(* LS Electric XG5000 project: InchingWalkThroughEX *)
(* PLC LSPLC *)
(* module base 0 slot 0: Input/Output Module:XEM-DN/DP32HP (DC 24V Input, Transistor Output, 32 Contacts) *)
(* module base 0 slot 1: Internal Positioning:XBF-PO06E (Open Collector Type, 6 Axis) *)

(* Comments on direct variables
%IX0.0.4	Jog FWD Ax1
%IX0.0.5	Jog REV Ax1
*)

PROGRAM Jog (* task: Scan Program *)
VAR
    Axis1_Inch_FWD : APM_INC;
    Axis1_Inch_FWD1 : XPM_INC;
    Axis1_Inch_REV : XPM_INC;
    Axis1_Jog_FWD : XPM_JOG;
    Axis1_Jog_REV : XPM_JOG;
    AXIS1_RST : XPM_RST;
    Axis1_RTP : XPM_RTP;
    Axis1_STP : XPM_STP;
END_VAR

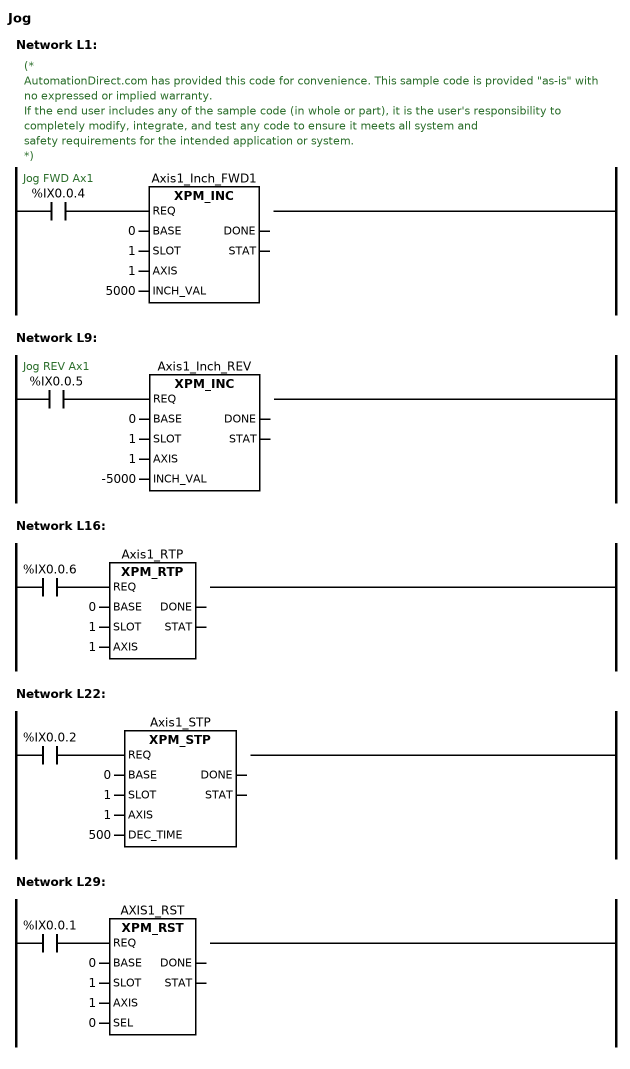
(* ( * / AutomationDirect.com has provided this code for convenience. This sample code is provided "as-is" with no expressed or implied warranty. / If the end user includes any of the sample code (in whole or part), it is the user's responsibility to completely modify, integrate, and test any code to ensure it meets all system and / safety requirements for the intended application or system. / * ) *)
(* Rung L1 *)
Axis1_Inch_FWD1(REQ := %IX0.0.4, BASE := 0, SLOT := 1, AXIS := 1, INCH_VAL := 5000);
(* Rung L9 *)
Axis1_Inch_REV(REQ := %IX0.0.5, BASE := 0, SLOT := 1, AXIS := 1, INCH_VAL := -5000);
(* Rung L16 *)
Axis1_RTP(REQ := %IX0.0.6, BASE := 0, SLOT := 1, AXIS := 1);
(* Rung L22 *)
Axis1_STP(REQ := %IX0.0.2, BASE := 0, SLOT := 1, AXIS := 1, DEC_TIME := 500);
(* Rung L29 *)
AXIS1_RST(REQ := %IX0.0.1, BASE := 0, SLOT := 1, AXIS := 1, SEL := 0);
END_PROGRAM